PROGRAM prgHeatPump
VAR
	fb_word_to_float	:FB_CV_WORD_TO_REAL_FLOAT;
	real_ProductionTemperatureOut		: REAL;									//{#lynus.ag#()}
	real_ProductionTemperatureIn		: REAL;									//{#lynus.ag#()}
	real_CompresorSuctionPressure		: REAL;									//{#lynus.ag#()}
	real_CompressorDischargePressure	: REAL;									//{#lynus.ag#()}
	real_DHWTemperature					: REAL;									//{#lynus.ag#()}
	real_OutdoorTemperature				: REAL;									//{#lynus.ag#()}
	real_BrineCircuitPressure			: REAL;									//{#lynus.ag#()}
	real_ProductionCircuitPressure		: REAL;									//{#lynus.ag#()}
	real_CompressorStartTempForDHW		: REAL;									//{#lynus.ag#()}
	real_COP							: REAL;									//{#lynus.ag#()}
	real_PF								: REAL;									//{#lynus.ag#()}
	real_CondensationTemperature		: REAL;									//{#lynus.ag#()}
	real_Superheat						: REAL;									//{#lynus.ag#()}
	real_ExpansionValvePosition			: REAL;									//{#lynus.ag#()}
	real_SetpointDHWBUS					: REAL;									//{#lynus.ag#()}
	real_BUSHeatingDG1Setpoint			: REAL;									//{#lynus.ag#()}
	real_BUSHeatingSG2Setpoint			: REAL;									//{#lynus.ag#()}
	real_BUSHeatingSG3Setpoint			: REAL;									//{#lynus.ag#()}
	real_BUSHeatingSG4Setpoint			: REAL;									//{#lynus.ag#()}
	real_BUSCoolingDG1Setpoint			: REAL;									//{#lynus.ag#()}
	real_BUSCoolingSG2Setpoint			: REAL;									//{#lynus.ag#()}
	real_BUSCoolingSG3Setpoint			: REAL;									//{#lynus.ag#()}
	real_BUSCoolingSG4Setpoint			: REAL;									//{#lynus.ag#()}
	real_SupplytemperatureSG2			: REAL;									//{#lynus.ag#()}
	real_SupplytemperatureSG3			: REAL;									//{#lynus.ag#()}
	real_SupplytemperatureSG4			: REAL;									//{#lynus.ag#()}
	real_DHWStarttemperature			: REAL;									//{#lynus.ag#()}
	real_Evaporationtemperature			: REAL;									//{#lynus.ag#()}
	real_Heatingbuffertanktemp			: REAL;									//{#lynus.ag#()}
	real_Coolingbuffertanktemp			: REAL;									//{#lynus.ag#()}
	real_EER							: REAL;									//{#lynus.ag#()}
	real_Compresordischargetemp			: REAL;									//{#lynus.ag#()}
	real_Surplusactivationsetpoint		: REAL;									//{#lynus.ag#()}
	real_Consumptionlimitsetpoint 		: REAL;									//{#lynus.ag#()}
	real_CompressorRPM					: REAL;									//{#lynus.ag#()}
	real_ScrollTemp						: REAL;									//{#lynus.ag#()}
	real_Invertertemperature			: REAL;									//{#lynus.ag#()}
	real_Powerconsumption				: REAL;									//{#lynus.ag#()}
	real_Condensationcapacity			: REAL;									//{#lynus.ag#()}

	real_Heatpumpstate					: REAL;									//{#lynus.ag#()}
	// 1=Off; 2=On; 3=Emergency; 0=Keyboard
	real_Workingprogram					: REAL;									//{#lynus.ag#()}
	// 1=Winter;2=Summer; 3=Mixed; 0=Keyboard
	real_BUS_DHWDemand					: REAL;									//{#lynus.ag#()}
	real_BUS_SG2Demand					: REAL;									//{#lynus.ag#()}
	real_BUS_SG3Demand					: REAL;									//{#lynus.ag#()}
	real_BUS_SG4Demand					: REAL;									//{#lynus.ag#()}
//	real_			: REAL;									//{#lynus.ag#()}
//	real_			: REAL;									//{#lynus.ag#()}
	
	bool_HP_Alarm					: BOOL;								//{#lynus.ag#()}
	bool_HP_BusControlEnable		: BOOL;								//{#lynus.ag#()}

	mTest: BOOL;

END_VAR

MODBUS_RTU_EcoForest();
IF MODBUS_RTU_EcoForest.structArrayModbusRTU[1].wArrayReceiveBuffer[10]<>0 THEN 	
	real_ProductionTemperatureOut 	:=INT_TO_REAL(WORD_TO_INT(MODBUS_RTU_EcoForest.structArrayModbusRTU[1].wArrayReceiveBuffer[2]))/10;
	real_ProductionTemperatureIn 	:=INT_TO_REAL(WORD_TO_INT(MODBUS_RTU_EcoForest.structArrayModbusRTU[1].wArrayReceiveBuffer[3]))/10;
	real_CompresorSuctionPressure 	:=INT_TO_REAL(WORD_TO_INT(MODBUS_RTU_EcoForest.structArrayModbusRTU[1].wArrayReceiveBuffer[5]))/10;
	real_CompressorDischargePressure:=int_to_real(word_to_int(MODBUS_RTU_EcoForest.structArrayModbusRTU[1].wArrayReceiveBuffer[6]))/10;
	real_DHWTemperature				:=int_to_real(word_to_int(MODBUS_RTU_EcoForest.structArrayModbusRTU[1].wArrayReceiveBuffer[7]))/10;
	real_OutdoorTemperature			:=int_to_real(word_to_int(MODBUS_RTU_EcoForest.structArrayModbusRTU[1].wArrayReceiveBuffer[10]))/10;
	real_BrineCircuitPressure		:=int_to_real(word_to_int(MODBUS_RTU_EcoForest.structArrayModbusRTU[1].wArrayReceiveBuffer[12]))/10;
	real_ProductionCircuitPressure	:=int_to_real(word_to_int(MODBUS_RTU_EcoForest.structArrayModbusRTU[1].wArrayReceiveBuffer[13]))/10;
	real_CompressorStartTempForDHW	:=int_to_real(word_to_int(MODBUS_RTU_EcoForest.structArrayModbusRTU[1].wArrayReceiveBuffer[14]))/10;
END_IF
IF (MODBUS_RTU_EcoForest.structArrayModbusRTU[2].wArrayReceiveBuffer[7])/10 <> 0 THEN	
	real_COP						:= INT_TO_REAL(WORD_TO_INT(MODBUS_RTU_EcoForest.structArrayModbusRTU[2].wArrayReceiveBuffer[7]))/10;	
	real_PF							:= INT_TO_REAL(WORD_TO_INT(MODBUS_RTU_EcoForest.structArrayModbusRTU[2].wArrayReceiveBuffer[8]))/10;
END_IF	
IF  (MODBUS_RTU_EcoForest.structArrayModbusRTU[3].wArrayReceiveBuffer[0])/10 <>0 THEN 	
	real_CondensationTemperature	:= INT_TO_REAL(WORD_TO_INT(MODBUS_RTU_EcoForest.structArrayModbusRTU[3].wArrayReceiveBuffer[0]))/10;	
END_IF	
IF (MODBUS_RTU_EcoForest.structArrayModbusRTU[4].wArrayReceiveBuffer[1])/10 <> 0 THEN
	real_Superheat					:= INT_TO_REAL(WORD_TO_INT(MODBUS_RTU_EcoForest.structArrayModbusRTU[4].wArrayReceiveBuffer[0]))/10;	
	real_ExpansionValvePosition		:= int_to_real(word_to_int(MODBUS_RTU_EcoForest.structArrayModbusRTU[4].wArrayReceiveBuffer[1]))/10;	
	real_SetpointDHWBUS				:= int_to_real(word_to_int(MODBUS_RTU_EcoForest.structArrayModbusRTU[4].wArrayReceiveBuffer[2]))/10;	
	real_BUSHeatingDG1Setpoint		:= int_to_real(word_to_int(MODBUS_RTU_EcoForest.structArrayModbusRTU[4].wArrayReceiveBuffer[3]))/10;	
	real_BUSHeatingSG2Setpoint		:= int_to_real(word_to_int(MODBUS_RTU_EcoForest.structArrayModbusRTU[4].wArrayReceiveBuffer[4]))/10;	
	real_BUSHeatingSG3Setpoint		:= int_to_real(word_to_int(MODBUS_RTU_EcoForest.structArrayModbusRTU[4].wArrayReceiveBuffer[5]))/10;	
	real_BUSHeatingSG4Setpoint		:= int_to_real(word_to_int(MODBUS_RTU_EcoForest.structArrayModbusRTU[4].wArrayReceiveBuffer[6]))/10;	
	real_BUSCoolingDG1Setpoint		:= int_to_real(word_to_int(MODBUS_RTU_EcoForest.structArrayModbusRTU[4].wArrayReceiveBuffer[7]))/10;	
	real_BUSCoolingSG2Setpoint		:= int_to_real(word_to_int(MODBUS_RTU_EcoForest.structArrayModbusRTU[4].wArrayReceiveBuffer[8]))/10;	
	real_BUSCoolingSG3Setpoint		:= int_to_real(word_to_int(MODBUS_RTU_EcoForest.structArrayModbusRTU[4].wArrayReceiveBuffer[9]))/10;	
	real_BUSCoolingSG4Setpoint		:= INT_TO_REAL(WORD_TO_INT(MODBUS_RTU_EcoForest.structArrayModbusRTU[4].wArrayReceiveBuffer[10]))/10;	
END_IF


IF (MODBUS_RTU_EcoForest.structArrayModbusRTU[7].wArrayReceiveBuffer[1])/10 <> 0 THEN 
	real_SupplytemperatureSG2		:= INT_TO_REAL(WORD_TO_INT(MODBUS_RTU_EcoForest.structArrayModbusRTU[7].wArrayReceiveBuffer[0]))/10;	
	real_SupplytemperatureSG3		:= int_to_real(word_to_int(MODBUS_RTU_EcoForest.structArrayModbusRTU[7].wArrayReceiveBuffer[1]))/10;	
	real_SupplytemperatureSG4		:= int_to_real(word_to_int(MODBUS_RTU_EcoForest.structArrayModbusRTU[7].wArrayReceiveBuffer[2]))/10;	
	real_DHWStarttemperature		:= int_to_real(word_to_int(MODBUS_RTU_EcoForest.structArrayModbusRTU[7].wArrayReceiveBuffer[3]))/10;	
	real_Evaporationtemperature		:= int_to_real(word_to_int(MODBUS_RTU_EcoForest.structArrayModbusRTU[7].wArrayReceiveBuffer[4]))/10;	
	real_Heatingbuffertanktemp		:= int_to_real(word_to_int(MODBUS_RTU_EcoForest.structArrayModbusRTU[7].wArrayReceiveBuffer[5]))/10;	
	real_Coolingbuffertanktemp		:= int_to_real(word_to_int(MODBUS_RTU_EcoForest.structArrayModbusRTU[7].wArrayReceiveBuffer[6]))/10;	
	real_EER						:= int_to_real(word_to_int(MODBUS_RTU_EcoForest.structArrayModbusRTU[7].wArrayReceiveBuffer[7]))/10;	
	real_Compresordischargetemp		:= int_to_real(word_to_int(MODBUS_RTU_EcoForest.structArrayModbusRTU[7].wArrayReceiveBuffer[8]))/10;	
END_IF

IF (MODBUS_RTU_EcoForest.structArrayModbusRTU[8].wArrayReceiveBuffer[0])/10 <> 0 THEN
	real_Surplusactivationsetpoint	:= INT_TO_REAL(WORD_TO_INT(MODBUS_RTU_EcoForest.structArrayModbusRTU[8].wArrayReceiveBuffer[0]))/10;	
	real_Consumptionlimitsetpoint	:= INT_TO_REAL(WORD_TO_INT(MODBUS_RTU_EcoForest.structArrayModbusRTU[8].wArrayReceiveBuffer[1]))/10;	
END_IF

IF MODBUS_RTU_EcoForest.structArrayModbusRTU[5].wArrayReceiveBuffer[3] <> 0 THEN		
	real_CompressorRPM 				:= INT_TO_REAL(WORD_TO_INT(MODBUS_RTU_EcoForest.structArrayModbusRTU[5].wArrayReceiveBuffer[0]));
	real_ScrollTemp					:= int_to_real(word_to_int(MODBUS_RTU_EcoForest.structArrayModbusRTU[5].wArrayReceiveBuffer[2]));
	real_Invertertemperature		:= int_to_real(word_to_int(MODBUS_RTU_EcoForest.structArrayModbusRTU[5].wArrayReceiveBuffer[3]));
END_IF

IF MODBUS_RTU_EcoForest.structArrayModbusRTU[6].wArrayReceiveBuffer[3] <> 0 THEN
	real_Powerconsumption			:= INT_TO_REAL(WORD_TO_INT(MODBUS_RTU_EcoForest.structArrayModbusRTU[6].wArrayReceiveBuffer[2]));		
	real_Condensationcapacity		:= INT_TO_REAL(WORD_TO_INT(MODBUS_RTU_EcoForest.structArrayModbusRTU[6].wArrayReceiveBuffer[3]));		
END_IF

IF MODBUS_RTU_EcoForest.structArrayModbusRTU[9].wArrayReceiveBuffer[8] <> 0 THEN // [8] = Start counter
	real_Heatpumpstate		:= INT_TO_REAL(WORD_TO_INT(MODBUS_RTU_EcoForest.structArrayModbusRTU[9].wArrayReceiveBuffer[0]));	
	real_Workingprogram		:= INT_TO_REAL(WORD_TO_INT(MODBUS_RTU_EcoForest.structArrayModbusRTU[9].wArrayReceiveBuffer[1]));	
	real_BUS_DHWDemand		:= INT_TO_REAL(WORD_TO_INT(MODBUS_RTU_EcoForest.structArrayModbusRTU[9].wArrayReceiveBuffer[2]));
	real_BUS_SG2Demand		:= INT_TO_REAL(WORD_TO_INT(MODBUS_RTU_EcoForest.structArrayModbusRTU[9].wArrayReceiveBuffer[4]));	
	real_BUS_SG3Demand		:= INT_TO_REAL(WORD_TO_INT(MODBUS_RTU_EcoForest.structArrayModbusRTU[9].wArrayReceiveBuffer[5]));	
	real_BUS_SG4Demand		:= INT_TO_REAL(WORD_TO_INT(MODBUS_RTU_EcoForest.structArrayModbusRTU[9].wArrayReceiveBuffer[6]));	
END_IF
	

bool_HP_Alarm 				:= WORD_TO_BOOL(MODBUS_RTU_EcoForest.structArrayModbusRTU[10].wArrayReceiveBuffer[0]);
bool_HP_BusControlEnable	:= WORD_TO_BOOL(MODBUS_RTU_EcoForest.structArrayModbusRTU[10].wArrayReceiveBuffer[3]);

//			:= INT_TO_REAL(WORD_TO_INT(MODBUS_RTU_EcoForest.structArrayModbusRTU[].wArrayReceiveBuffer[]));	
//			:= INT_TO_REAL(WORD_TO_INT(MODBUS_RTU_EcoForest.structArrayModbusRTU[].wArrayReceiveBuffer[]));

END_PROGRAM

(* stored: Version 1.1.0.1, ProductVersion 3.1.4024.12
   POU prgHeatPump: Id {4b08ab89-193c-4965-952f-17b12cf78ea8}, SpecialFunc None *)
